(* PLC project OOP_Curso, Beckhoff Automation GmbH TwinCAT PLC Control 3.5.13.21 *)
(* stored: creationDateTime 2023-10-28T13:22:48.2872608, modificationDateTime 2023-10-28T13:22:48.2970201 *)

(*
### This sample project contains the following elements.

- FB_UML_SC:		This FB represents a simulation to save a text as XML or text format, and to publish it afterwards to a client and to a master.
					The underlying state machine is implemented with the help of UML State Chart.
					
					The behavior is not really programmed.
					Only the wrapper/basic structure of the state machine is implemented. 
						
					Each time, when an ENTRY/DO/EXIT action is called, a correspondent counter variable is increased.

- Visualization:	The visu shows the state of the counters, so that you can see how often an ENTRY/DO/EXIT action has been called. 
					You can use the buttons to switch between the states.
*)
PROGRAM _32_MAIN
VAR
	fbUmlSC	: FB_UML_SC;
END_VAR

            fbUmlSC();
          
END_PROGRAM

FUNCTION_BLOCK FB_UML_SC
VAR
	// Transition condition
	bInitFinished				: BOOL;
	bUseXmlFormat				: BOOL;
	bAllInfoCopiedToFile		: BOOL;
	bSendToMasterFinished		: BOOL;
	bSendToClientFinished		: BOOL;
	
	// Counters
	nCounterInit				: INT;
	nCounterSaveInitSettings	: INT;
	nCounterClearXml			: INT;
	nCounterFillXml				: INT;
	nCounterSaveXml				: INT;
	nCounterClearText			: INT;
	nCounterFillText			: INT;
	nCounterSaveText			: INT;
	nCounterGetMasterID			: INT;
	nCounterGetClientID			: INT;
	nCounterSendToMaster		: INT;
	nCounterSendToClient		: INT;
	
	// Debugging
	bMasterFirst				: BOOL;
	bClientFirst				: BOOL;
END_VAR

            
          

METHOD PROTECTED ClearTextFile
VAR_INPUT
END_VAR
                  nCounterClearText := nCounterClearText + 1;
                
END_METHOD

METHOD PROTECTED ClearXmlFile
VAR_INPUT
END_VAR
                  nCounterClearXml := nCounterClearXml + 1;
                
END_METHOD

METHOD PROTECTED FillTextFile
VAR_INPUT
END_VAR
                  nCounterFillText := nCounterFillText + 1;
                
END_METHOD

METHOD PROTECTED FillXmlFile
VAR_INPUT
END_VAR
                  nCounterFillXml := nCounterFillXml + 1;
                
END_METHOD

METHOD PROTECTED GetClientID
VAR_INPUT
END_VAR
                  nCounterGetClientID := nCounterGetClientID + 1;

IF NOT bMasterFirst THEN
	bClientFirst := TRUE;
END_IF
                
END_METHOD

METHOD PROTECTED GetMasterID
VAR_INPUT
END_VAR
                  nCounterGetMasterID := nCounterGetMasterID + 1;

IF NOT bClientFirst THEN
	bMasterFirst := TRUE;
END_IF
                
END_METHOD

METHOD PROTECTED Init
VAR_INPUT
END_VAR
                  nCounterInit := nCounterInit + 1;
                
END_METHOD

METHOD PROTECTED SaveInitSettings
VAR_INPUT
END_VAR
                  nCounterSaveInitSettings := nCounterSaveInitSettings + 1;

bInitFinished 			:= FALSE;
bAllInfoCopiedToFile 	:= FALSE;
bSendToClientFinished 	:= FALSE;
bSendToMasterFinished	:= FALSE;
bMasterFirst			:= FALSE;
bClientFirst			:= FALSE;
                
END_METHOD

METHOD PROTECTED SaveTextFile
VAR_INPUT
END_VAR
                  nCounterSaveText := nCounterSaveText + 1;
                
END_METHOD

METHOD PROTECTED SaveXmlFile
VAR_INPUT
END_VAR
                  nCounterSaveXml := nCounterSaveXml + 1;
                
END_METHOD

METHOD PROTECTED SendFileToClient
VAR_INPUT
END_VAR
                  nCounterSendToClient := nCounterSendToClient + 1;
                
END_METHOD

METHOD PROTECTED SendFileToMaster
VAR_INPUT
END_VAR
                  nCounterSendToMaster := nCounterSendToMaster + 1;
                
END_METHOD
END_FUNCTION_BLOCK

{attribute 'no-analysis' := ''}
{attribute 'reduced_bp_set' := ''}
PROGRAM Kaffemaschine
VAR
	bMakeCoffee: BOOL := FALSE;
	bShutDown: BOOL := FALSE;
	bPowerUp: BOOL := FALSE;
	nGrind: INT := 0;
	nHeat: INT := 20;
	nFoam: INT := 0;
	{attribute 'implicit_state_chart_struct' := ''}
	UML_SC_Kaffemaschine: _UML_SC_7cc42eb0dc6d4e02ab5b1296bec80ed6;
	{attribute 'implicit_state_chart_struct' := ''}
	UML_SC_ActHeat: _UML_SC_9e3c3d30f6c84991be9f932f948dff00;
END_VAR

            
          

ACTION ActDo:
                nGrind := nGrind + 10;
              
END_ACTION

ACTION ActEntry:
                
              
END_ACTION

ACTION ActFoam:
                nFoam := nFoam + 5;
              
END_ACTION

ACTION ActHeat:
                
              
END_ACTION

ACTION ActShutdown:
                bShutDown := FALSE;
bPowerUp := FALSE;
              
END_ACTION

ACTION CoffeeReady:
                bMakeCoffee := FALSE;
nGrind := 0;
nHeat := 20;
nFoam := 0;
              
END_ACTION
END_PROGRAM
